// TIA Portal V17 export
// export: Created 2026-05-13T16:51:30.84957Z, ExportSetting WithDefaults, DisplayName Totally Integrated Automation Portal, DisplayVersion V17 Update 4, DisplayName TIA Portal Openness, DisplayVersion V17 Update 4, DisplayName TIA Portal Version Control Interface, DisplayVersion V17, DisplayName SINAMICS Startdrive Advanced, DisplayVersion V17, DisplayName SINAMICS Startdrive G130, G150, S120, S150, SINAMICS MV, S210, DisplayVersion V17, DisplayName SINAMICS Startdrive G110M, G120, G120C, G120D, G120P, G115D, DisplayVersion V17, DisplayName STEP 7 Professional, DisplayVersion V17 Update 4, DisplayName STEP 7 Safety, DisplayVersion V17, DisplayName WinCC Professional, DisplayVersion V17 Update 4
GraphicList "火焰"  ListRange=Decimal, Mode=Simple
  GraphicListEntry   EntryType=SingleValue, Picture=火焰1
  GraphicListEntry   EntryType=SingleValue, From=1, To=1, Picture=火焰2
  GraphicListEntry   EntryType=SingleValue, From=2, To=2, Picture=火焰3
  GraphicListEntry   EntryType=SingleValue, From=3, To=3, Picture=火焰4
  GraphicListEntry   EntryType=SingleValue, From=4, To=4, Picture=火焰5
